FUNCTION FN_MemoryClear
VAR_INPUT
	destAddr: PVOID;
	Len: UDINT;
END_VAR
VAR
	NULL: BYTE:= 0;
	i: ULINT;
END_VAR


	FOR i := 0 TO (Len-1) BY 1 DO
		MEMCPY(destAddr:= destAddr + i, srcAddr:= ADR(NULL), n:= 1);				
	END_FOR

END_FUNCTION

(* stored: Version 1.1.0.1, ProductVersion 3.1.4024.13
   POU FN_MemoryClear: Id {52b7d7fc-56ef-4523-95ac-807eab11f276}, SpecialFunc None *)
